// Mitsubishi GX Works2 project: PLC과제   PLC: Q00J
// 1학기

PROGRAM MAIN
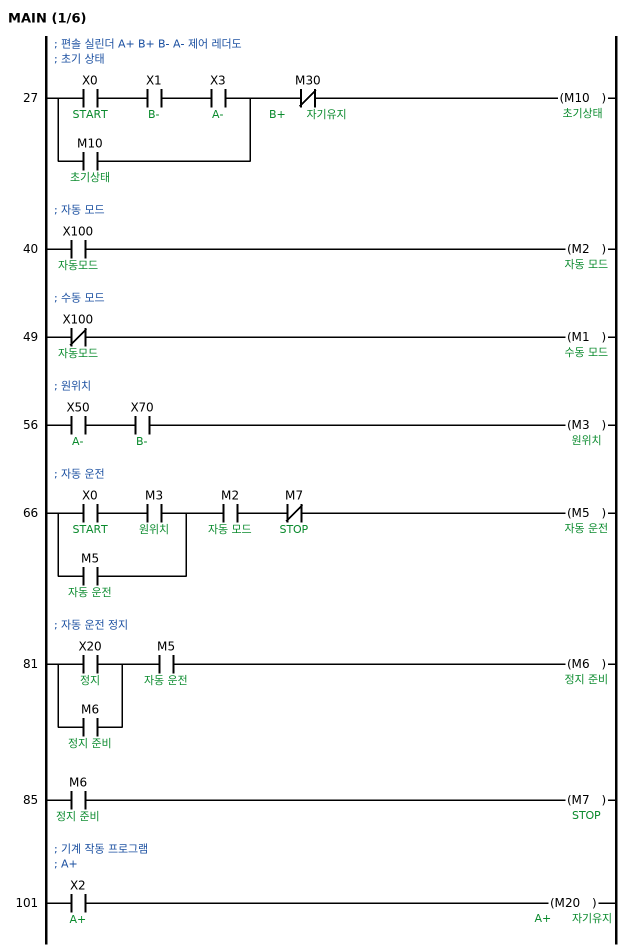
; 편솔 실린더 A+ B+ B- A- 제어 레더도
; 초기 상태
27    LD      X0  ; START
      AND     X1  ; B-
      AND     X3  ; A-
      OR      M10  ; 초기상태
      ANI     M30  ; B+      자기유지
      OUT     M10  ; 초기상태
; 자동 모드
40    LD      X100  ; 자동모드
      OUT     M2  ; 자동 모드
; 수동 모드
49    LDI     X100  ; 자동모드
      OUT     M1  ; 수동 모드
; 원위치
56    LD      X50  ; A-
      AND     X70  ; B-
      OUT     M3  ; 원위치
; 자동 운전
66    LD      X0  ; START
      AND     M3  ; 원위치
      OR      M5  ; 자동 운전
      AND     M2  ; 자동 모드
      ANI     M7  ; STOP
      OUT     M5  ; 자동 운전
; 자동 운전 정지
81    LD      X20  ; 정지
      OR      M6  ; 정지 준비
      AND     M5  ; 자동 운전
      OUT     M6  ; 정지 준비
85    LD      M6  ; 정지 준비
      OUT     M7  ; STOP
; 기계 작동 프로그램
; A+
101   LD      X2  ; A+
      OUT     M20  ; A+      자기유지
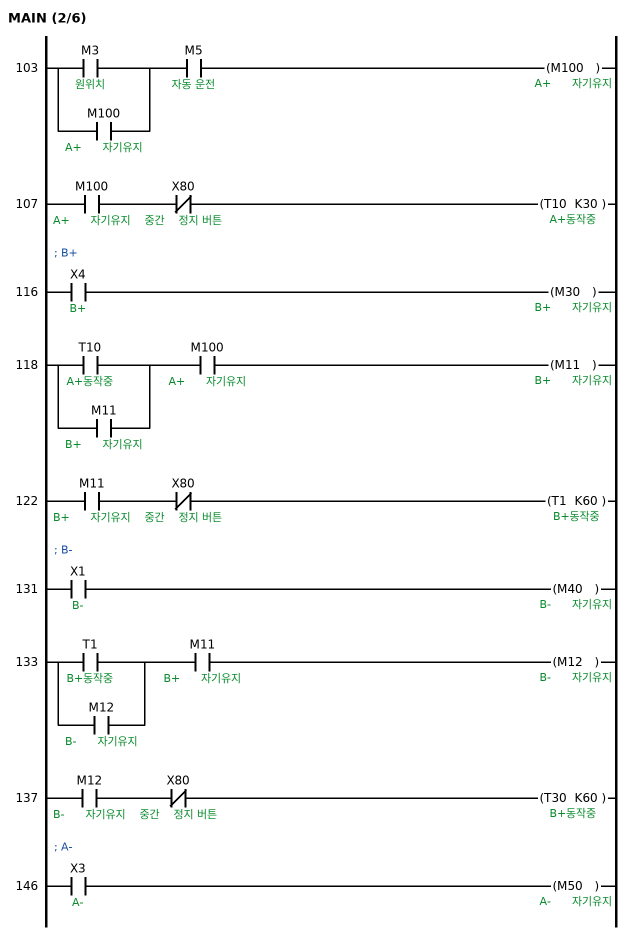
103   LD      M3  ; 원위치
      OR      M100  ; A+      자기유지
      AND     M5  ; 자동 운전
      OUT     M100  ; A+      자기유지
107   LD      M100  ; A+      자기유지
      ANI     X80  ; 중간    정지 버튼
      OUT     T10 K30  ; A+동작중
; B+
116   LD      X4  ; B+
      OUT     M30  ; B+      자기유지
118   LD      T10  ; A+동작중
      OR      M11  ; B+      자기유지
      AND     M100  ; A+      자기유지
      OUT     M11  ; B+      자기유지
122   LD      M11  ; B+      자기유지
      ANI     X80  ; 중간    정지 버튼
      OUT     T1 K60  ; B+동작중
; B-
131   LD      X1  ; B-
      OUT     M40  ; B-      자기유지
133   LD      T1  ; B+동작중
      OR      M12  ; B-      자기유지
      AND     M11  ; B+      자기유지
      OUT     M12  ; B-      자기유지
137   LD      M12  ; B-      자기유지
      ANI     X80  ; 중간    정지 버튼
      OUT     T30 K60  ; B+동작중
; A-
146   LD      X3  ; A-
      OUT     M50  ; A-      자기유지
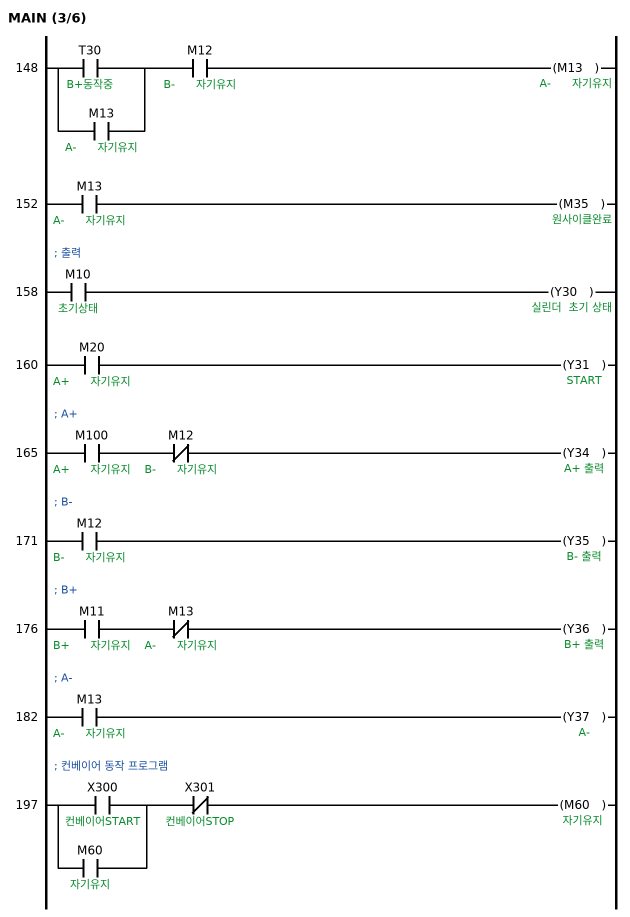
148   LD      T30  ; B+동작중
      OR      M13  ; A-      자기유지
      AND     M12  ; B-      자기유지
      OUT     M13  ; A-      자기유지
152   LD      M13  ; A-      자기유지
      OUT     M35  ; 원사이클완료
; 출력
158   LD      M10  ; 초기상태
      OUT     Y30  ; 실린더  초기 상태
160   LD      M20  ; A+      자기유지
      OUT     Y31  ; START
; A+
165   LD      M100  ; A+      자기유지
      ANI     M12  ; B-      자기유지
      OUT     Y34  ; A+ 출력
; B-
171   LD      M12  ; B-      자기유지
      OUT     Y35  ; B- 출력
; B+
176   LD      M11  ; B+      자기유지
      ANI     M13  ; A-      자기유지
      OUT     Y36  ; B+ 출력
; A-
182   LD      M13  ; A-      자기유지
      OUT     Y37  ; A-
; 컨베이어 동작 프로그램
197   LD      X300  ; 컨베이어START
      OR      M60  ; 자기유지
      ANI     X301  ; 컨베이어STOP
      OUT     M60  ; 자기유지
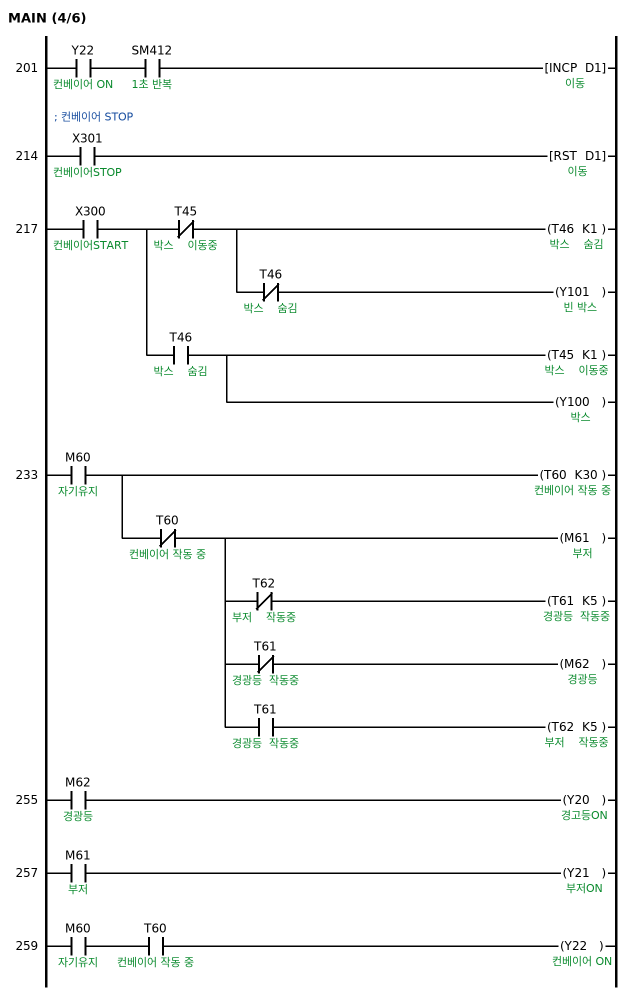
201   LD      Y22  ; 컨베이어 ON
      AND     SM412  ; 1초 반복
      INCP    D1  ; 이동
; 컨베이어 STOP
214   LD      X301  ; 컨베이어STOP
      RST     D1  ; 이동
217   LD      X300  ; 컨베이어START
      MPS
      ANI     T45  ; 박스    이동중
      OUT     T46 K1  ; 박스    숨김
      ANI     T46  ; 박스    숨김
      OUT     Y101  ; 빈 박스
      MPP
      AND     T46  ; 박스    숨김
      OUT     T45 K1  ; 박스    이동중
      OUT     Y100  ; 박스
233   LD      M60  ; 자기유지
      OUT     T60 K30  ; 컨베이어 작동 중
      ANI     T60  ; 컨베이어 작동 중
      OUT     M61  ; 부저
      MPS
      ANI     T62  ; 부저    작동중
      OUT     T61 K5  ; 경광등  작동중
      MRD
      ANI     T61  ; 경광등  작동중
      OUT     M62  ; 경광등
      MPP
      AND     T61  ; 경광등  작동중
      OUT     T62 K5  ; 부저    작동중
255   LD      M62  ; 경광등
      OUT     Y20  ; 경고등ON
257   LD      M61  ; 부저
      OUT     Y21  ; 부저ON
259   LD      M60  ; 자기유지
      AND     T60  ; 컨베이어 작동 중
      OUT     Y22  ; 컨베이어 ON
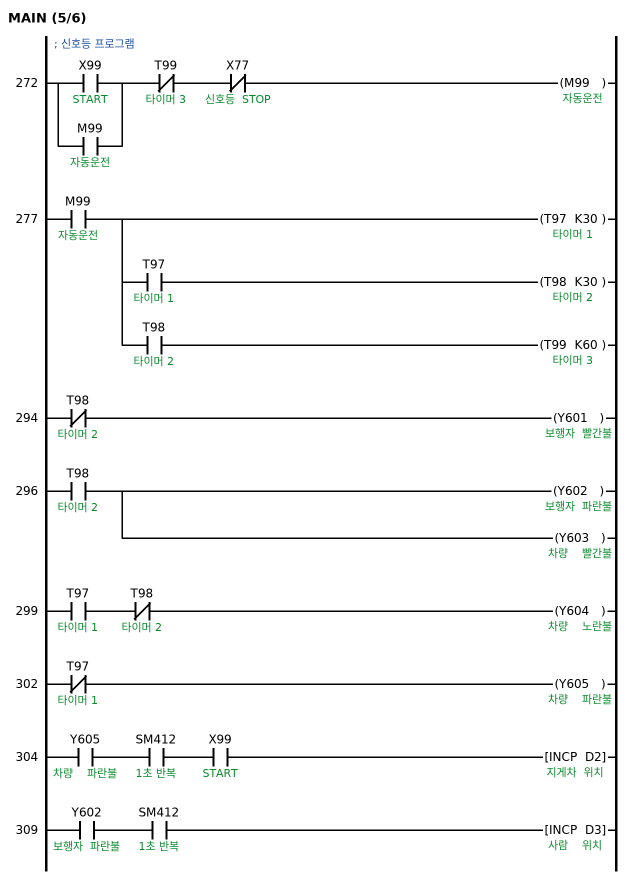
; 신호등 프로그램
272   LD      X99  ; START
      OR      M99  ; 자동운전
      ANI     T99  ; 타이머 3
      ANI     X77  ; 신호등  STOP
      OUT     M99  ; 자동운전
277   LD      M99  ; 자동운전
      OUT     T97 K30  ; 타이머 1
      MPS
      AND     T97  ; 타이머 1
      OUT     T98 K30  ; 타이머 2
      MPP
      AND     T98  ; 타이머 2
      OUT     T99 K60  ; 타이머 3
294   LDI     T98  ; 타이머 2
      OUT     Y601  ; 보행자  빨간불
296   LD      T98  ; 타이머 2
      OUT     Y602  ; 보행자  파란불
      OUT     Y603  ; 차량    빨간불
299   LD      T97  ; 타이머 1
      ANI     T98  ; 타이머 2
      OUT     Y604  ; 차량    노란불
302   LDI     T97  ; 타이머 1
      OUT     Y605  ; 차량    파란불
304   LD      Y605  ; 차량    파란불
      AND     SM412  ; 1초 반복
      AND     X99  ; START
      INCP    D2  ; 지게차  위치
309   LD      Y602  ; 보행자  파란불
      AND     SM412  ; 1초 반복
      INCP    D3  ; 사람    위치
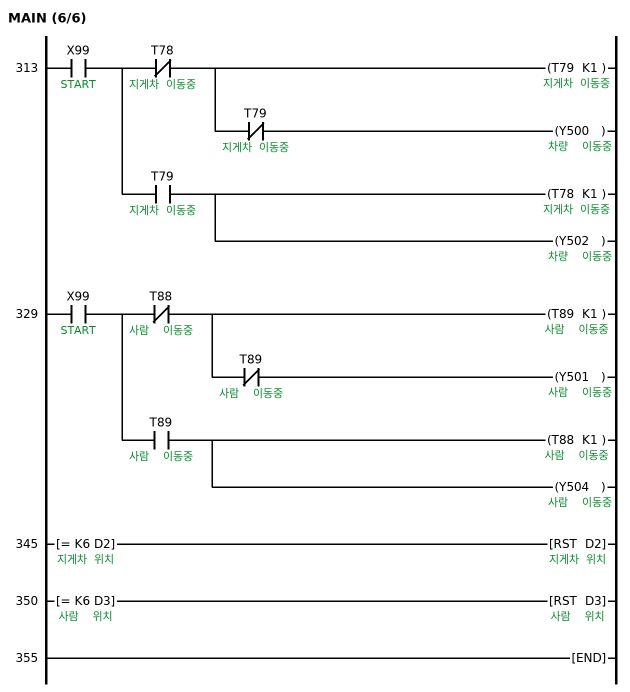
313   LD      X99  ; START
      MPS
      ANI     T78  ; 지게차  이동중
      OUT     T79 K1  ; 지게차  이동중
      ANI     T79  ; 지게차  이동중
      OUT     Y500  ; 차량    이동중
      MPP
      AND     T79  ; 지게차  이동중
      OUT     T78 K1  ; 지게차  이동중
      OUT     Y502  ; 차량    이동중
329   LD      X99  ; START
      MPS
      ANI     T88  ; 사람    이동중
      OUT     T89 K1  ; 사람    이동중
      ANI     T89  ; 사람    이동중
      OUT     Y501  ; 사람    이동중
      MPP
      AND     T89  ; 사람    이동중
      OUT     T88 K1  ; 사람    이동중
      OUT     Y504  ; 사람    이동중
345   LD=     K6 D2  ; 지게차  위치
      RST     D2  ; 지게차  위치
350   LD=     K6 D3  ; 사람    위치
      RST     D3  ; 사람    위치
355   END
END_PROGRAM
